// Mitsubishi GX Works2 project: 17+   PLC: FX3G

// task Task_01 (event TRUE, interval 0, priority 31): POU_01

PROGRAM POU_01
VAR
  wstep : INT;
  ton1 : TON;
  ton2 : TON;
  ton3 : TON;
  ton5 : TON;
  ton4 : TON;
  ton6 : TON;
  ton7 : TON;
  ton8 : TON;
  ton9 : TON;
  ton10 : TON;
  ton12 : TON;
  ton11 : TON;
  ton13 : TON;
  ton14 : TON;
  ton15 : TON;
END_VAR
IF M8002 THEN
	wstep := 0;
END_IF;

IF NOT M1 THEN
	wstep := 0;
END_IF;

CASE wstep OF
	0:
		ZRST(TRUE, M2, M99);
		IF M1 THEN
			wstep := 20;
		END_IF;
		
	20:
		M13 := TRUE;
		M15 := FALSE;
		M23 := TRUE;
		M25 := FALSE;
		M35 := TRUE;
		M45 := TRUE;
		ton1(IN := NOT ton1.Q, PT := T#5s);
		IF ton1.Q THEN
			wstep := 21;
		END_IF;
		
	21:
		M12 := TRUE;
		M13 := FALSE;
		M22 := TRUE;
		M23 := FALSE;
		ton2(IN := NOT ton2.Q, PT := T#5s);
		IF ton2.Q THEN
			wstep := 22;
		END_IF;		
		
	22:
		M11 := TRUE;
		M12 := FALSE;
		M21 := TRUE;
		M22 := FALSE;
		ton3(IN := NOT ton3.Q, PT := T#5s);
		IF ton3.Q THEN
			wstep := 23;
		END_IF;
		
	23:
		M11 := M8013;
		M21 := NOT M8013;
		ton4(IN := NOT ton4.Q, PT := T#3s);
		IF ton4.Q THEN
			wstep := 24;
		END_IF;		
		
	24:
		M11 := FALSE;
		M14 := TRUE;
		M21 := FALSE;
		M24 := TRUE;
		ton5(IN := NOT ton5.Q, PT := T#5s);
		IF ton5.Q THEN
			wstep := 25;
		END_IF;		
		
	25:
		M14 := FALSE;
		M15 := TRUE;
		M24 := FALSE;
		M25 := TRUE;
		ton6(IN := NOT ton6.Q, PT := T#3s);
		IF ton6.Q THEN
			wstep := 26;
		END_IF;	
	
	26:
		M33 := TRUE;
		M35 := FALSE;
		M43 := TRUE;
		M45 := FALSE;
		ton7(IN := NOT ton7.Q, PT := T#5s);
		IF ton7.Q THEN
			wstep := 27;
		END_IF;
		
	27:
		M33 := FALSE;
		M32 := TRUE;
		M43 := FALSE;
		M42 := TRUE;
		ton8(IN := NOT ton8.Q, PT := T#5s);
		IF ton8.Q THEN
			wstep := 28;
		END_IF;		
		
	28:
		M32 := FALSE;
		M31 := TRUE;
		M42 := FALSE;
		M41 := TRUE;
		ton9(IN := NOT ton9.Q, PT := T#5s);
		IF ton9.Q THEN
			wstep := 29;
		END_IF;			
		
	29:
		M31 := M8013;
		M41 := NOT M8013;
		ton10(IN := NOT ton10.Q, PT := T#3s);
		IF ton10.Q THEN
			wstep := 30;
		END_IF;		
		
	30:
		M31 := FALSE;
		M34 := TRUE;
		M41 := FALSE;
		M44 := TRUE;
		ton11(IN := NOT ton11.Q, PT := T#3s);
		IF ton11.Q THEN
			wstep := 31;
		END_IF;	
		
	31:
		M34 := FALSE;
		M35 := TRUE;
		M44 := FALSE;
		M45 := TRUE;
		ton12(IN := NOT ton12.Q, PT := T#3s);
		IF ton12.Q THEN
			wstep := 20;
		END_IF;			
			
END_CASE;
END_PROGRAM
